{attribute addProperty BoxType "EL1262-0000-0002"}
{attribute addProperty Id "Ch1_CycleCountAT %I*Ch1_CycleCount_2F207C3C1620Ch1_InputAT %I*ARRAY[0..9] OF Ch1_Input_FD9B961D80100GapAT %I*EMPTY_STRUCTURE000Ch2_CycleCountAT %I*Ch2_CycleCount_7D759C541620Ch2_InputAT %I*ARRAY[0..9] OF Ch2_Input_E3B70EF680100Gap_1AT %I*EMPTY_STRUCTURE000NextSync1TimeAT %I*NextSync1Time_EAC4272D3240WcStateAT %I*WcState_F855686C1620InfoDataAT %I*InfoData_7231B2DD80100"}
{attribute addProperty CRC "3584440036"}
{attribute addProperty SizeInBites "320"}
{attribute addProperty SizeInBytes "40"}
TYPE EL1262_0572C526 :
STRUCT
	{attribute addProperty Name "Ch1_CycleCount"}
	Ch1_CycleCount : Ch1_CycleCount_2F207C3C;
	{attribute addProperty Name "Ch1_Input"}
	Ch1_Input : ARRAY[0..9] OF Ch1_Input_FD9B961D;
	{attribute addProperty Name "Gap"}
	Gap : EMPTY_STRUCTURE;
	{attribute addProperty Name "Ch2_CycleCount"}
	Ch2_CycleCount : Ch2_CycleCount_7D759C54;
	{attribute addProperty Name "Ch2_Input"}
	Ch2_Input : ARRAY[0..9] OF Ch2_Input_E3B70EF6;
	{attribute addProperty Name "Gap_1"}
	Gap_1 : EMPTY_STRUCTURE;
	{attribute addProperty Name "NextSync1Time"}
	NextSync1Time : NextSync1Time_EAC4272D;
	{attribute addProperty Name "WcState"}
	WcState : WcState_F855686C;
	{attribute addProperty Name "InfoData"}
	InfoData : InfoData_7231B2DD;
END_STRUCT
END_TYPE

(* stored: Version 1.2.0.0, ProductVersion 3.1.4024.9
   DUT EL1262_0572C526: Id {5a1ee59d-e941-41e5-970e-ee9894c11666} *)
